PROGRAM Motor_Aixs02_X
VAR
END_VAR

// NETWORK 1

END_PROGRAM

(* stored: Version 1.1.0.1, ProductVersion 3.1.4024.15
   POU Motor_Aixs02_X: Id {d9213bc4-148a-4239-a203-38f23f33a9e8}, SpecialFunc None *)
